(* IEC 61131-3 sources: plcassist-cli/packages/volt-lsp-iec/test-corpus/pro2193/Device/Plc Logic/Application/99 Library/Function Blocks/Modules, 9 files *)

(* ---- LockFB.fb ---- *)
// Use the TEST_AND_SET operator to ensure exclusive access.
{attribute 'no_explicit_call' := 'No need to call this FB. Only the methods are used'}
{attribute 'monitoring_display' := 'currentLockHolder'}
FUNCTION_BLOCK LockFB
VAR
	dwSynch							: DWORD;		// Lock object
	currentLockHolder				: STRING(80);	// Name of the module that is currently locking this FB
	currentLockHolderIsWithoutLock	: BOOL;
END_VAR
VAR_OUTPUT
	callCounter						: UDINT;
END_VAR

END_FUNCTION_BLOCK

// Force releasing the lock
METHOD ForceRelease
Release(currentLockHolder);
END_METHOD

// Release the lock by the current lock holder
METHOD Release : BOOL
VAR_INPUT
	locker		: STRING(80);		// The module that is releasing the lock
END_VAR
IF locker <> currentLockHolder THEN
	RETURN;
END_IF

IF locker <> '' OR dwSynch <> 0 THEN
	LogPlc.Debug(CONCAT5('Lock released by: ', locker, ', lock duration: ', TO_STRING(callCounter), ' PLC cycles'));
END_IF

dwSynch							:= 0;		// The DWORD must be reset to release the lock
currentLockHolder				:= '';		// Clear name of locker
currentLockHolderIsWithoutLock	:= FALSE;
callCounter						:= 0;

Release							:= TRUE;
END_METHOD

// Request a lock. Returns false if the lock is already taken by someone else.
METHOD Request : BOOL
VAR_INPUT
	locker		: STRING(80);		// The module that is requesting the lock
END_VAR
IF currentLockHolder = locker THEN		// Check if already locked by locker
	Request := TRUE;					// Locking succeeded
ELSIF TEST_AND_SET(dwSynch) = 0 THEN	// Write the 1 and read the old value at the same time; Result of 0 means no other task is currently locking this FB
	currentLockHolder := locker;		// Save name of locker
	LogPlc.Debug(CONCAT('Lock granted to: ', locker));
	Request := TRUE;					// Locking succeeded
ELSIF currentLockHolderIsWithoutLock THEN
	currentLockHolder := locker;		// Save name of locker
	LogPlc.Debug(CONCAT('Lock stolen by: ', locker));
	Request := TRUE;					// Locking succeeded
ELSE
	Request := FALSE;					// Locking failed. Allready locked by someone else.
END_IF

IF Request THEN
	callCounter := callCounter + 1;
END_IF
END_METHOD

// Request a lock without actually locking. Use if a command should be overruled by a second command.
{attribute 'obsolete' := 'Do not use! Method makes no sense. See below for discussion'}
METHOD RequestWithoutLock : BOOL
VAR_INPUT
	locker		: STRING(80);		// The module that is requesting the lock
END_VAR

// locking without actually locking makes no sense to me!
// Just NOT lock a command if you don't need a lock.
// If we really need it we could add optional bool parameter to Request method: WeakLock or something
// Stefan 3-7-25
IF currentLockHolder = locker THEN		// Check if already locked by locker
	RequestWithoutLock := TRUE;			// Locking succeeded
ELSIF TEST_AND_SET(dwSynch) = 0 THEN	// Write the 1 and read the old value at the same time; Result of 0 means no other task is currently locking this FB
	currentLockHolder := locker;		// Save name of locker
	LogPlc.Debug(CONCAT('Lock granted to: ', locker));
	currentLockHolderIsWithoutLock := TRUE;
	RequestWithoutLock := TRUE;			// Locking succeeded
ELSIF currentLockHolderIsWithoutLock THEN
	currentLockHolder := locker;		// Save name of locker
	LogPlc.Debug(CONCAT('Lock stolen by: ', locker));
	RequestWithoutLock := TRUE;			// Locking succeeded
ELSE
	RequestWithoutLock := FALSE;		// Locking failed. Allready locked by someone else.
END_IF

IF RequestWithoutLock THEN
	callCounter := callCounter + 1;
END_IF
END_METHOD

// Return true the first cycle that the lock is granted.
PROPERTY PUBLIC FirstCall : BOOL

// No monitoring attribute because property is only high for 1 cycle.
GET
VAR
END_VAR
FirstCall := callCounter = 1;
END_GET
END_PROPERTY

// Return true when a lock is active
{attribute 'monitoring':='call'}
PROPERTY PUBLIC IsLocked : BOOL
GET
VAR
END_VAR
IsLocked := currentLockHolder <> '';
END_GET
END_PROPERTY

(* ---- ModuleBaseHardwareFB.fb ---- *)
// Modules that react to EStop and Stop events from the machine
{attribute 'symbol' := 'none'}
FUNCTION_BLOCK PUBLIC ABSTRACT ModuleBaseHardwareFB
EXTENDS ModuleRegisterableFB
IMPLEMENTS IModuleBase, IModuleWithCommandLock
VAR
	CommandLock					: LockFB;		// Internal lock. Lock hardware unit when a command is active
	ProcessCommandLock			: LockFB;		// External lock from the process. So a process can claim a hardware unit for itself
END_VAR

SUPER^();

Alarms();	// Handle custom alarms that are not defined in the FB's called in Cyclic()

END_FUNCTION_BLOCK

METHOD PROTECTED Alarms
END_METHOD

// Command to reset the module (Statemachine to zero state) in case of E-Stop
METHOD PUBLIC EStop : BOOL	// Returns true when drives are in standstill

(* Command to reset the module (Statemachine to zero state) in case of E-Stop

Add code here to handle emergency stops. For example:

// Reset the state of the unit.
State := MyUnit_State.None;

// Stop the servo drive
Drive.Stop(TRUE);

// Reset all cylinders and outputs
SomeCylinder.Reset();
SomeOtherOutput.Reset();

// Reset all vacuums with a helper function
VacuumResetAll(Vacuum);

// Does this module have a servo drive? Then you can return true when the drive has braked to standstill
EStop := Drive.Standstill OR NOT Drive.AxisEnabled;
// Else, just return true.
EStop := TRUE;

 *)
CommandLock.ForceRelease();
ProcessCommandLock.ForceRelease();

EStop := TRUE;
END_METHOD

// Force releasing the lock
METHOD LockForceRelease
ProcessCommandLock.ForceRelease();
END_METHOD

// Release the lock by the current lock holder
METHOD PUBLIC LockRelease : BOOL
VAR_INPUT
	locker		: STRING(80);		// The module that is releasing the lock
END_VAR
LockRelease		:= ProcessCommandLock.Release(locker);
END_METHOD

// Request a lock. Returns false if the lock is already taken by someone else.
METHOD PUBLIC LockRequest : BOOL
VAR_INPUT
	locker		: STRING(80);		// The module that is requesting the lock
END_VAR
LockRequest		:= ProcessCommandLock.Request(locker);
END_METHOD

// Command to stop a module (Statemachine to zero state)
METHOD PUBLIC Stop : BOOL	// Returns true when drives are in standstill
CommandLock.ForceRelease();
ProcessCommandLock.ForceRelease();

Stop := TRUE;
END_METHOD

(* ---- ModuleManagerFB.fb ---- *)
// Function block to register all modules in the program. So its no longer needed to manually fill an array in the SER program.
{attribute 'no_explicit_call' := 'Do not call this FB. This is just a place to store data about regestered modules.'}
{attribute 'no_assign'}
FUNCTION_BLOCK FINAL ModuleManagerFB
IMPLEMENTS IModuleManager
VAR_OUTPUT
	baseModules				: ARRAY[1..GVL_Constants.MaxNumberOfModules] OF IModuleBase;
	baseModulesCount		: UINT;

	startableModules		: ARRAY[1..GVL_Constants.MaxNumberOfStartableModules] OF IModuleStartable;
	startableModulesCount	: UINT;

	resettableModules		: ARRAY[1..GVL_Constants.MaxNumberOfResettableModules] OF IModuleResettable;
	resettableModulesCount	: UINT;

	servoDrives				: ARRAY[1..GVL_Constants.MaxNumberOfServoDrives] OF IServoDrive;
	servoDrivesCount		: UINT;

	gates					: ARRAY[1..GVL_Constants.MaxNumberOfGates] OF ISafetyGate;
	gatesCount				: UINT;

END_VAR
VAR
	{attribute 'hide'}	_name					: STRING(12);									// Name of module manager
	{attribute 'hide'}	_moduleHandler			: L_IMHP.L_IMHP_ModuleHandler :=				// Lenze module handler
						(
							Layer				:= L_IMHP_Layer.Process_Control,
							CompType			:= L_IMHP_ComponentType.GeneralMachineModule
						);
END_VAR

END_FUNCTION_BLOCK

//FB_Init is always available implicitly and it is used primarily for initialization.
//The return value is not evaluated. For a specific influence, you can also declare the
//methods explicitly and provide additional code there with the standard initialization
//code. You can evaluate the return value.
METHOD FB_Init: BOOL
VAR_INPUT
	bInitRetains	: BOOL;							// TRUE: the retain variables are initialized (reset warm / reset cold)
	bInCopyCode		: BOOL;							// TRUE: the instance will be copied to the copy code afterward (online change)

	name			: STRING(12);					// Give name of module manager (For example SER or BFU)
END_VAR
THIS^._name						:= name;
THIS^._moduleHandler.CompName	:= name;
END_METHOD

METHOD PRIVATE LogMessage
VAR_INPUT
	moduleName		: STRING(12);
	selUnRegister	: BOOL;
	index			: UINT;
	module			: IAbleToRegister;
END_VAR
LogPlc.Debug(
	CONCAT9(
		Name,
		': ',
		moduleName,
		' module ',
		TO_STRING(index),
		SEL(selUnRegister, ' registered: ', ' unregistered: '),
		module.InstanceName,
		SEL(module.MemoryAddress = '', ', Address: ', ''),
		module.MemoryAddress
	)
);
END_METHOD

// Registers a module
METHOD Register : BOOL
VAR_INPUT
	thingToRegister	: IAbleToRegister;
END_VAR
VAR
	baseModule		: IModuleBase;
	startableModule	: IModuleStartable;
	resettableModule: IModuleResettable;
	servoDrive		: IServoDrive;
	gate			: ISafetyGate;

	thingMatchedAnyInterface : BOOL;
END_VAR
IF thingToRegister = 0 THEN
	LogPlc.Fatal('Null reference exception! Interface does not exist.');
	RETURN;
END_IF

IF __QUERYINTERFACE(thingToRegister, baseModule) THEN
	IF baseModulesCount = GVL_Constants.MaxNumberOfModules THEN
		LogPlc.Fatal(CONCAT('Register Full! Module NOT registered: ', thingToRegister.InstanceName));
	ELSE
		thingMatchedAnyInterface				:= TRUE;
		Increment.AnyInt(baseModulesCount);
		baseModules[baseModulesCount]			:= baseModule;
		LogMessage('Base', FALSE, baseModulesCount, thingToRegister);
	END_IF
END_IF

IF __QUERYINTERFACE(thingToRegister, startableModule) THEN
	IF startableModulesCount = GVL_Constants.MaxNumberOfStartableModules THEN
		LogPlc.Fatal(CONCAT('Startable Register Full! Module NOT registered: ', thingToRegister.InstanceName));
	ELSE
		thingMatchedAnyInterface				:= TRUE;
		Increment.AnyInt(startableModulesCount);
		startableModules[startableModulesCount]	:= startableModule;
		LogMessage('Startable', FALSE, startableModulesCount, thingToRegister);
	END_IF
END_IF

IF __QUERYINTERFACE(thingToRegister, resettableModule) THEN
	IF resettableModulesCount = GVL_Constants.MaxNumberOfResettableModules THEN
		LogPlc.Fatal(CONCAT('Resettable Register Full! Module NOT registered: ', thingToRegister.InstanceName));
	ELSE
		thingMatchedAnyInterface				:= TRUE;
		Increment.AnyInt(resettableModulesCount);
		resettableModules[resettableModulesCount] := resettableModule;
		LogMessage('Resettable', FALSE, resettableModulesCount, thingToRegister);
	END_IF
END_IF

IF __QUERYINTERFACE(thingToRegister, servoDrive) THEN
	IF servoDrivesCount = GVL_Constants.MaxNumberOfServoDrives THEN
		LogPlc.Fatal(CONCAT('Servodrive Register Full! Module NOT registered: ', thingToRegister.InstanceName));
	ELSE
		thingMatchedAnyInterface				:= TRUE;
		Increment.AnyInt(servoDrivesCount);
		servoDrives[servoDrivesCount]			:= servoDrive;
		LogMessage('Servo', FALSE, servoDrivesCount, thingToRegister);
	END_IF
END_IF

IF __QUERYINTERFACE(thingToRegister, gate) THEN
	IF gatesCount = GVL_Constants.MaxNumberOfGates THEN
		LogPlc.Fatal(CONCAT('Gate Register Full! Module NOT registered: ', thingToRegister.InstanceName));
	ELSE
		thingMatchedAnyInterface				:= TRUE;
		Increment.AnyInt(gatesCount);
		gates[gatesCount]						:= gate;
		LogMessage('Gate', FALSE, gatesCount, thingToRegister);
	END_IF
END_IF

IF NOT thingMatchedAnyInterface THEN
	LogPlc.Fatal(Concat('Unable to register module: ', thingToRegister.InstanceName));	// Please add a handler for this kind of interface
END_IF

Register := TRUE;
END_METHOD

// Unregisters a module
METHOD Unregister : BOOL
VAR_INPUT
	thingToRegister	: IAbleToRegister;
END_VAR
VAR
	i				: UINT;
	moduleIndex		: UINT;
	baseModule		: IModuleBase;
	startableModule	: IModuleStartable;
	resettableModule: IModuleResettable;
	servoDrive		: IServoDrive;
	gate			: ISafetyGate;
	thingMatchedAnyInterface : BOOL;
END_VAR
IF thingToRegister = 0 THEN
	LogPlc.Fatal('Null reference exception! Interface does not exist.');
	RETURN;
END_IF

// Check if the current interface is of type: module
IF __QUERYINTERFACE(thingToRegister, baseModule) THEN
	FOR i := 1 TO GVL_Constants.MaxNumberOfModules DO
		IF baseModule = baseModules[i] THEN		// Find the module in the register
			moduleIndex := i;				// Store location where it was found
			baseModules[i] := 0;			// Clear the reference
			baseModulesCount := baseModulesCount - 1;	// Decrease count
			LogMessage('Base', TRUE, moduleIndex, thingToRegister);
			EXIT;
		END_IF
	END_FOR
	// Move all references in the register one place up, so there are no gaps in the array.
	IF moduleIndex > 0 AND moduleIndex < GVL_Constants.MaxNumberOfModules THEN
		FOR i := moduleIndex TO GVL_Constants.MaxNumberOfModules - 1 DO
			baseModules[i] := baseModules[i + 1];
			IF baseModules[i + 1] = 0 THEN
				EXIT;
			END_IF
		END_FOR
	END_IF
	thingMatchedAnyInterface := TRUE;
	moduleIndex := 0;
END_IF

IF __QUERYINTERFACE(thingToRegister, startableModule) THEN
	FOR i := 1 TO GVL_Constants.MaxNumberOfStartableModules DO
		IF startableModule = startableModules[i] THEN
			moduleIndex := i;
			startableModules[i] := 0;
			startableModulesCount := startableModulesCount - 1;
			LogMessage('Startable', TRUE, moduleIndex, thingToRegister);
			EXIT;
		END_IF
	END_FOR
	IF moduleIndex > 0 AND moduleIndex < GVL_Constants.MaxNumberOfStartableModules THEN
		FOR i := moduleIndex TO GVL_Constants.MaxNumberOfStartableModules - 1 DO
			startableModules[i] := startableModules[i + 1];
			IF startableModules[i + 1] = 0 THEN
				EXIT;
			END_IF
		END_FOR
	END_IF
	thingMatchedAnyInterface := TRUE;
	moduleIndex := 0;
END_IF

IF __QUERYINTERFACE(thingToRegister, resettableModule) THEN
	FOR i := 1 TO GVL_Constants.MaxNumberOfResettableModules DO
		IF resettableModule = resettableModules[i] THEN
			moduleIndex := i;
			resettableModules[i] := 0;
			resettableModulesCount := resettableModulesCount - 1;
			LogMessage('Resettable', TRUE, moduleIndex, thingToRegister);
			EXIT;
		END_IF
	END_FOR
	IF moduleIndex > 0 AND moduleIndex < GVL_Constants.MaxNumberOfResettableModules THEN
		FOR i := moduleIndex TO GVL_Constants.MaxNumberOfResettableModules - 1 DO
			resettableModules[i] := resettableModules[i + 1];
			IF resettableModules[i + 1] = 0 THEN
				EXIT;
			END_IF
		END_FOR
	END_IF
	thingMatchedAnyInterface := TRUE;
	moduleIndex := 0;
END_IF

IF __QUERYINTERFACE(thingToRegister, servoDrive) THEN
	FOR i := 1 TO GVL_Constants.MaxNumberOfServoDrives DO
		IF servoDrive = servoDrives[i] THEN
			moduleIndex := i;
			servoDrives[i] := 0;
			servoDrivesCount := servoDrivesCount - 1;
			LogMessage('Servo', TRUE, moduleIndex, thingToRegister);
			EXIT;
		END_IF
	END_FOR
	IF moduleIndex > 0 AND moduleIndex < GVL_Constants.MaxNumberOfServoDrives THEN
		FOR i := moduleIndex TO GVL_Constants.MaxNumberOfServoDrives - 1 DO
			servoDrives[i] := servoDrives[i + 1];
			IF servoDrives[i + 1] = 0 THEN
				EXIT;
			END_IF
		END_FOR
	END_IF
	thingMatchedAnyInterface := TRUE;
	moduleIndex := 0;
END_IF

IF __QUERYINTERFACE(thingToRegister, gate) THEN
	FOR i := 1 TO GVL_Constants.MaxNumberOfGates DO
		IF gate = gates[i] THEN
			moduleIndex := i;
			gates[i] := 0;
			gatesCount := gatesCount - 1;
			LogMessage('Gate', TRUE, moduleIndex, thingToRegister);
			EXIT;
		END_IF
	END_FOR
	IF moduleIndex > 0 AND moduleIndex < GVL_Constants.MaxNumberOfGates THEN
		FOR i := moduleIndex TO GVL_Constants.MaxNumberOfGates - 1 DO
			gates[i] := gates[i + 1];
			IF gates[i + 1] = 0 THEN
				EXIT;
			END_IF
		END_FOR
	END_IF
	thingMatchedAnyInterface := TRUE;
	moduleIndex := 0;
END_IF

IF NOT thingMatchedAnyInterface THEN
	LogPlc.Fatal(Concat('Unable to unregister module: ', thingToRegister.InstanceName));	// Please add a handler for this kind of interface
END_IF

Unregister := TRUE;
END_METHOD

PROPERTY PUBLIC ModuleHandler : L_IMHP.L_IMHP_IModuleHandler
GET
VAR
END_VAR
ModuleHandler	:= _moduleHandler;
END_GET
END_PROPERTY

PROPERTY PUBLIC Name : STRING(12)
GET
VAR
END_VAR
Name	:= _name;

// This does not work because CompName has no Getter. Maybe change in the future when Lenze changes library
// Name	:= _moduleHandler.CompName;
END_GET
END_PROPERTY

(* ---- ModuleRegisterableFB.fb ---- *)
// Module registers itself with central module manager. Also implements Lenze module manager
{attribute 'reflection'}
{attribute 'monitoring_display' := '_instanceName'}
{attribute 'symbol' := 'none'}
FUNCTION_BLOCK PUBLIC ABSTRACT ModuleRegisterableFB
IMPLEMENTS IAbleToRegister
VAR
	ModuleManager				: IModuleManager;				// Location of module manager where this module is stored
	ModuleHandler				: L_IMHP.L_IMHP_ModuleHandler;	// Lenze module handler (No need to call this FB)

	{attribute 'hide'}
	{attribute 'no_copy'}
	_instanceNo					: UINT;				// Private backing field for instance number (start from 1)
	{attribute 'instance-path'}
	{attribute 'noinit'}
	{attribute 'hide'}
	_instanceName				: STRING(80);		// Private backing field for instance name (automatically generated by compiler)

	{attribute 'no_copy'}
	ModuleParent				: L_IMHP.L_IMHP_IModuleHandler;

	{attribute 'hide'}
	{attribute 'init_on_onlchange'}
	_initialized				: BOOL	:= FALSE;	// Is high when init is done
END_VAR
VAR_STAT
	moduleCurrentlyExecuting	: STRING(80);		// For debugging: In case of exception check this string to see what module is currently executing
END_VAR

IF NOT _initialized THEN
	_initialized := TRUE;
	Initialize();
END_IF

stu.StrCpyA(
	pBuffer		:= ADR(moduleCurrentlyExecuting),
	iBufferSize	:= SIZEOF(moduleCurrentlyExecuting),
	pStr		:= ADR(_instanceName)
	);

Cyclic();	// Do stuff every PLC cycle (like instantiate all fbs needed in the module).

END_FUNCTION_BLOCK

METHOD PROTECTED Cyclic
END_METHOD

//FB_Exit must be implemented explicitly. If there is an implementation, then the
//method is called before the controller removes the code of the function block instance
//(implicit call). The return value is not evaluated.
METHOD FB_Exit: BOOL
VAR_INPUT
	bInCopyCode: BOOL;  // TRUE: the exit method is called in order to leave the instance which will be copied afterwards (online change).
END_VAR
IF THIS^.ModuleManager <> 0 THEN
	THIS^.ModuleManager.Unregister(THIS^);
END_IF

THIS^.ModuleParent	:= 0;
END_METHOD

//FB_Init is always available implicitly and it is used primarily for initialization.
//The return value is not evaluated. For a specific influence, you can also declare the
//methods explicitly and provide additional code there with the standard initialization
//code. You can evaluate the return value.
METHOD FB_Init: BOOL
VAR_INPUT
	bInitRetains	: BOOL;							// TRUE: the retain variables are initialized (reset warm / reset cold)
	bInCopyCode		: BOOL;							// TRUE: the instance will be copied to the copy code afterward (online change)

	instanceNo		: UINT;
	moduleManager	: IModuleManager;				// Give location of module manager (can be different for SER or BFU)
	moduleParent	: L_IMHP.L_IMHP_IModuleHandler;	// (Optional) Give parent of this module. Use zero to use SER or BFU as parent.
END_VAR
THIS^.ModuleManager		:= moduleManager;

IF moduleManager = 0 THEN
	LogPlc.Info(CONCAT(_instanceName, ' has no module manager to register to. Is this intended?'));
ELSE
	moduleManager.Register(THIS^);		// Register this module with the central module manager.
END_IF

IF moduleParent <> 0 THEN
	THIS^.ModuleParent	:= moduleParent;
ELSIF moduleManager <> 0 THEN
	THIS^.ModuleParent	:= moduleManager.ModuleHandler;
END_IF

// Set instance number
IF instanceNo = 0 THEN
	LogPlc.Fatal(CONCAT(_instanceName, ' has instanceNo 0. Use instanceNo > 0.'));
END_IF

_instanceNo				:= instanceNo;

ParseInstanceName(ADR(_instanceName));

ModuleHandler.CompName	:= InstanceName;
ModuleHandler.Layer		:= L_IMHP_Layer.Tech_Application;
ModuleHandler.CompType	:= L_IMHP_ComponentType.GeneralMachineModule;

// Warning: Only when module is of CompType = MachineModule or GeneralMachineModule, are active alarms kicked up to the parent module!
END_METHOD

METHOD PROTECTED Initialize
ModuleHandler.SetParent(
					ModuleHandlerParent	:= ModuleParent,
					RelationShip		:= L_IMHP.L_IMHP_RelationshipID.ApplicationView);
END_METHOD

// Automatically generated name of the instance
{attribute 'monitoring':='call'}
PROPERTY PUBLIC InstanceName : STRING(80)
GET
VAR
END_VAR
InstanceName := _instanceName;
END_GET
END_PROPERTY

// Instance number, the number of the module or unit (start from 1)
{attribute 'monitoring':='call'}
PROPERTY PUBLIC InstanceNo : UINT

// Note: this number does not have to be unique for each module...
GET
VAR
END_VAR
InstanceNo := _instanceNo;
END_GET
END_PROPERTY

// Location of the FB in memory (for debugging)
{attribute 'monitoring':='call'}
PROPERTY PUBLIC MemoryAddress : STRING(8)
GET
VAR
END_VAR
{IF defined (IsSimulationMode)}
	MemoryAddress := DWORD_TO_HEXSTRING(TO_DWORD(ADR(THIS^)));
{ELSE}
	MemoryAddress := '';
{END_IF}
END_GET
END_PROPERTY

(* ---- ModuleResettableFB.fb ---- *)
// Generic variables that all modules use
{attribute 'symbol' := 'none'}
FUNCTION_BLOCK PUBLIC ABSTRACT ModuleResettableFB
EXTENDS ModuleBaseHardwareFB
IMPLEMENTS IModuleResettable
VAR
	{attribute 'hide'}
	{attribute 'no_copy'}
	_resetConditions			: ARRAY[1..2] OF IModuleResettable;
END_VAR

SUPER^();

END_FUNCTION_BLOCK

//FB_Init is always available implicitly and it is used primarily for initialization.
//The return value is not evaluated. For a specific influence, you can also declare the
//methods explicitly and provide additional code there with the standard initialization
//code. You can evaluate the return value.
{attribute 'analysis' := '-33'}
METHOD FB_Init: BOOL
VAR_INPUT
	bInitRetains	: BOOL;							// TRUE: the retain variables are initialized (reset warm / reset cold)
	bInCopyCode		: BOOL;							// TRUE: the instance will be copied to the copy code afterward (online change)

	instanceNo		: UINT;							// Handled in ModuleRegisterableFB.FB_Init method
	moduleManager	: IModuleManager;				// Handled in ModuleRegisterableFB.FB_Init method
	moduleParent	: L_IMHP.L_IMHP_IModuleHandler;	// Handled in ModuleRegisterableFB.FB_Init method

	resetCondition1	: IModuleResettable;
	resetCondition2	: IModuleResettable;
END_VAR
_resetConditions[1]	:= resetCondition1;
_resetConditions[2]	:= resetCondition2;
END_METHOD

// Command to reset the module. Servodrives are homed.
METHOD PUBLIC ABSTRACT Reset : BOOL	// Returns true when homing done
END_METHOD

// The order in which the modules are homed.
{attribute 'monitoring':='call'}
PROPERTY PUBLIC ResetCondition1 : IModuleResettable
GET
VAR
END_VAR
ResetCondition1	:= _resetConditions[1];
END_GET
END_PROPERTY

// The order in which the modules are homed.
{attribute 'monitoring':='call'}
PROPERTY PUBLIC ResetCondition2 : IModuleResettable
GET
VAR
END_VAR
ResetCondition2	:= _resetConditions[2];
END_GET
END_PROPERTY

(* ---- ModuleWithBrakedServoBaseFB.fb ---- *)
// Extra variables for modules that have a servo drive
{attribute 'symbol' := 'none'}
FUNCTION_BLOCK PUBLIC ABSTRACT ModuleWithBrakedServoBaseFB
EXTENDS ModuleWithServoBaseFB
VAR_INPUT
	ButtonReleaseBrake			: PushButtonLedFB;
END_VAR
VAR
	{attribute 'symbol' := 'read'}	DriveBrakeLogic				: ServoDriveBrakeLogicFB;
END_VAR

SUPER^(
	AxisRef				:= AxisRef,
	DataBrink			:= DataBrink,
	coveredDistance		:= coveredDistance,
);

ButtonReleaseBrake();

DriveBrakeLogic(
	AxisRef				:= AxisRef,
	xBrakeReleaseIn		:= ButtonReleaseBrake.buttonInput);

END_FUNCTION_BLOCK

(* ---- ModuleWithServoBaseFB.fb ---- *)
// Extra variables for modules that have a servo drive
{attribute 'symbol' := 'none'}
FUNCTION_BLOCK PUBLIC ABSTRACT ModuleWithServoBaseFB
EXTENDS ModuleResettableFB
IMPLEMENTS IModuleManualControlEnabled
VAR_INPUT
	xEnableServoDrive			: BOOL;
	xQuickStop					: BOOL;
END_VAR
VAR_IN_OUT
	AxisRef						: L_MC1P.AXIS_REF;
	DataBrink					: DataBrinkType;
	coveredDistance				: UDINT;
END_VAR
VAR
	{attribute 'symbol' := 'read'}	Drive						: ServoDriveFB
	(
		instanceNo		:= 1,
		moduleManager	:= ModuleManager,
		moduleParent	:= ModuleHandler,
	);

	// Forward alarms of children (ServoDriveFB) to parent
	ForwardSeverity				: L_IE1P.L_IE1P_ForwardSeverity;

	// Manual control of servo drive is enabled from outside this module
	externalManualServoControlEnabled		: BOOL;
	// Manual control of servo drive is enabled from inside the module
	internalManualServoControlEnabled		: BOOL := TRUE;

	ManualControlIsBlockedWarning			: ARRAY[1..6] OF SetErrorFB;

END_VAR

SUPER^();

Drive(
	globalSpeedOverride			:= PersistentVars.usiGlobalSERSpeed,
	globalSpeedOverrideEnable	:= ,
	rSetManualSpeed				:= 5,
	xGlobalReset				:= GlobalVars.Reset,
	xEnableDrive				:= xEnableServoDrive,
	xQuickStop					:= xQuickStop,
	manualControlEnabled		:= SER.ManualControlEnabled
								AND Drive.AxisEnabled
								AND externalManualServoControlEnabled
								AND internalManualServoControlEnabled
								AND PNOZMulti2.xHoldToRunButton,
	servoJogMode				:= HMI.servoJogMode,
	AxisRef						:= AxisRef,
	DataBrink					:= DataBrink,
	coveredDistance				:= coveredDistance);

ForwardSeverity(
	xEnable						:= TRUE,
	ModuleHandler				:= ModuleHandler,
	xForwardFromChildModules	:= TRUE,
	xDisableForwardToParent		:= ,
	xBusy						=> ,
	xError						=> ,
	eErrorID					=> );

ManualControlIsBlockedWarning[1](
	moduleHandler	:= ModuleHandler,
	textRefId		:= General_Unit_Errors,
	errorId			:= 6,
	alarmCondition	:= Drive.manualControlIsBlocked AND NOT SER.ManualControlEnabled,
	alarmDelay		:= 0.0,
	severity		:= enumErrorSeverity.Warning_Lock,
	reaction		:= enumErrorReaction.No_reaction);

ManualControlIsBlockedWarning[2](
	moduleHandler	:= ModuleHandler,
	textRefId		:= General_Unit_Errors,
	errorId			:= 7,
	alarmCondition	:= Drive.manualControlIsBlocked AND NOT Drive.AxisEnabled,
	alarmDelay		:= 0.0,
	severity		:= enumErrorSeverity.Warning_Lock,
	reaction		:= enumErrorReaction.No_reaction);

ManualControlIsBlockedWarning[3](
	moduleHandler	:= ModuleHandler,
	textRefId		:= General_Unit_Errors,
	errorId			:= 8,
	alarmCondition	:= Drive.manualControlIsBlocked AND NOT externalManualServoControlEnabled,
	alarmDelay		:= 0.0,
	severity		:= enumErrorSeverity.Warning_Lock,
	reaction		:= enumErrorReaction.No_reaction);

ManualControlIsBlockedWarning[4](
	moduleHandler	:= ModuleHandler,
	textRefId		:= General_Unit_Errors,
	errorId			:= 9,
	alarmCondition	:= Drive.manualControlIsBlocked AND NOT internalManualServoControlEnabled,
	alarmDelay		:= 0.0,
	severity		:= enumErrorSeverity.Warning_Lock,
	reaction		:= enumErrorReaction.No_reaction);

ManualControlIsBlockedWarning[5](
	moduleHandler	:= ModuleHandler,
	textRefId		:= General_Unit_Errors,
	errorId			:= 10,
	alarmCondition	:= Drive.manualControlIsBlocked AND NOT PNOZMulti2.xHoldToRunButton,
	alarmDelay		:= 0.0,
	severity		:= enumErrorSeverity.Warning_Lock,
	reaction		:= enumErrorReaction.No_reaction);

ManualControlIsBlockedWarning[6](
	moduleHandler	:= ModuleHandler,
	textRefId		:= General_Unit_Errors,
	errorId			:= 11,
	alarmCondition	:= Drive.manualControlIsBlocked AND Drive.AxisBasicControl.xInternalControlActive,
	alarmDelay		:= 0.0,
	severity		:= enumErrorSeverity.Warning_Lock,
	reaction		:= enumErrorReaction.No_reaction);

END_FUNCTION_BLOCK

METHOD PROTECTED Initialize
SUPER^.Initialize();

Drive.config.axisBlockedAlarmMaxTorque	:= 0.5;
END_METHOD

// Manual control of hardware is enabled from external context
{attribute 'monitoring':='call'}
PROPERTY ExternalManualControlEnabled : BOOL
SET
VAR
END_VAR
externalManualServoControlEnabled := ExternalManualControlEnabled;
END_SET
END_PROPERTY

(* ---- ModuleWithStateFB.fb ---- *)
// Modules that have a state (Processes). Keep a history with StateMachineHistoryFB
{attribute 'symbol' := 'none'}
FUNCTION_BLOCK PUBLIC ABSTRACT ModuleWithStateFB
EXTENDS ModuleRegisterableFB
IMPLEMENTS IModuleBase
VAR
	CommandLock					: LockFB;		// Internal lock. Lock hardware unit when a command is active (check if we can remove this!! Processes do not need locks ?? SR)

	{attribute 'symbol' := 'read'}	State	: StateMachineHistoryFB(instanceName:= InstanceName);		// Call this FB in Cyclic() in your Process module!

	{attribute 'hide'}	noProgramWarningBusy		: BIT;
	{attribute 'hide'}	noProgramWarningDone		: BIT;
END_VAR

SUPER^();

noProgramWarningDone R= NOT noProgramWarningBusy;
noProgramWarningBusy := FALSE;

// Execute state machine of module
Execute();

END_FUNCTION_BLOCK

METHOD PROTECTED ABSTRACT Cyclic

// Modules with a State must have a Cyclic method: to call State FB
END_METHOD

// Command to reset the module (Statemachine to zero state) in case of E-Stop
METHOD PUBLIC ABSTRACT EStop : BOOL	// Returns true when drives are in standstill

(* Command to reset the module (Statemachine to zero state) in case of E-Stop

Add code here to handle emergency stops. For example:

// Reset the state of the unit.
State := MyUnit_State.None;

// Stop the servo drive
Drive.Stop(TRUE);

// Reset all cylinders and outputs
SomeCylinder.Reset();
SomeOtherOutput.Reset();

// Reset all vacuums with a helper function
VacuumResetAll(Vacuum);

// Does this module have a servo drive? Then you can return true when the drive has braked to standstill
EStop := Drive.Standstill OR NOT Drive.AxisEnabled;
// Else, just return true.
EStop := TRUE;

 *)
END_METHOD

// After a state change, this method is called to execute the current state
METHOD PROTECTED ABSTRACT Execute
END_METHOD

// Here is the State Machine for the default exchangeset
METHOD PROTECTED ABSTRACT Execute_Sequence1
END_METHOD

// Logs a warning in the PLC log when there is a module that has not defined a program for an exchange set.
METHOD PROTECTED ShowNoProgramWarning
// Only write the log message once, the first time the method is executed.
IF NOT noProgramWarningDone THEN
	LogPlc.Warn(CONCAT3(InstanceName, ': No program for: ', TO_STRING(PersistentVars.RecipeVars.ActiveExchangeSet)));
END_IF

noProgramWarningBusy := TRUE;
noProgramWarningDone := TRUE;
END_METHOD

// Command to stop a module (Statemachine to zero state)
METHOD PUBLIC ABSTRACT Stop : BOOL	// Returns true when drives are in standstill
END_METHOD

(* ---- StateMachineHistoryFB.fb ---- *)
{attribute 'symbol' := 'none'}
FUNCTION_BLOCK INTERNAL FINAL StateMachineHistoryFB
EXTENDS MonitoringAddLogBase
VAR_INPUT
	{attribute 'symbol' := 'read'}	actState			: DINT;
END_VAR
VAR_OUTPUT
	StateHistory				: ARRAY[0..HistorySize] OF StateHistoryItemType;	// StateHistory[0] holds previous state
END_VAR
VAR//VISU
	{attribute 'symbol' := 'read'}	timeActive			: REAL;
	{attribute 'symbol' := 'read'}	timeIdle			: REAL;
	{attribute 'symbol' := 'read'}	durationInState		: REAL;						// Duration how long the current state is active.
	{attribute 'symbol' := 'read'}	actStateColor		: enumColorList;			// Color of active tile in HMI
END_VAR
VAR
	{attribute 'hide'}		i							: INT;
	{attribute 'hide'}		prevState					: DINT			:= GVL_Constants.DintSmallest;
	{attribute 'hide'}		timeLastStateTransition		: TIME_OF_DAY	:= TimeSettings.todNow;
	{attribute 'hide'}		instanceName				: STRING(80);
	{attribute 'hide'}		_stateChanged				: BOOL;

	{attribute 'hide'}		CycleTimeActive				: MeasureTime;				// Measure cycle times of this module
	{attribute 'hide'}		CycleTimeIdle				: MeasureTime;				// Measure cycle times of this module
	{attribute 'hide'}		measureDuration				: MeasureTime;

	timeout1_Warn_Delay			: REAL			:= 5.0;						// Color tile with warning color when state takes this long
	timeout2_Error_Delay		: REAL			:= 10.0;					// Color tile with error color when state takes this long
	timeout3_Fatal_Delay		: REAL			:= 15.0;					// Color tile with fatal color when state takes this long
	timeout1_Warn_Color			: enumColorList	:= enumColorList.Yellow;	// Warning color for tile
	timeout2_Error_Color		: enumColorList	:= enumColorList.Orange;	// Error color for tile
	timeout3_Fatal_Color		: enumColorList	:= enumColorList.Red;		// Fatal color for tile
END_VAR
VAR CONSTANT
	HistorySize					: INT := 19;
END_VAR

// Measure cycle times
timeIdle		:= CycleTimeActive.Measure(	In := actState < 10);
timeActive		:= CycleTimeIdle.Measure(	In := actState >= 10);
durationInState	:= measureDuration.Measure(	In := TRUE);	// Measure the duration how long the current step is active. Give the tile a color when it takes too long.

// Set color for tiles in HMI
IF actState < 10 THEN		// States 0 - 9 are idle states. Machine can stay in these states without timeouts
	actStateColor	:= enumColorList.Lime;
ELSIF durationInState > timeout3_Fatal_Delay THEN
	actStateColor	:= timeout3_Fatal_Color;
ELSIF durationInState > timeout2_Error_Delay THEN
	actStateColor	:= timeout2_Error_Color;
ELSIF durationInState > timeout1_Warn_Delay THEN
	actStateColor	:= timeout1_Warn_Color;
ELSE
	actStateColor	:= enumColorList.Lime;
END_IF

_stateChanged		:= FALSE;

// Check if act state is different than previous state
IF actState = prevState THEN
	RETURN;
END_IF

// Save a history of states
FOR i := HistorySize TO 1 BY -1 DO
	StateHistory[i]	:= StateHistory[i-1];
END_FOR

StateHistory[0].stateNumber			:= prevState;
StateHistory[0].durationInState		:= durationInState;
StateHistory[0].timeEnterState		:= timeLastStateTransition;
StateHistory[0].timeExitState		:= TimeSettings.todNow;

measureDuration.Measure(In := FALSE);
durationInState := 0;

// Save the time of the last state change
timeLastStateTransition	:= TimeSettings.todNow;

IF GlobalVars.EnableLoggingAllStateChanges THEN
	LogPlc.Info(CONCAT5(instanceName, ' changed state: ', TO_STRING(prevState), ' -> ', TO_STRING(actState)));
END_IF

// Output data to monitoring system (optional)
CallAddLogLINT(actState);

// Save previous state
prevState			:= actState;
_stateChanged		:= TRUE;

END_FUNCTION_BLOCK

//FB_Init is always available implicitly and it is used primarily for initialization.
//The return value is not evaluated. For a specific influence, you can also declare the
//methods explicitly and provide additional code there with the standard initialization
//code. You can evaluate the return value.
METHOD FB_Init: BOOL
VAR_INPUT
	bInitRetains: BOOL; // TRUE: the retain variables are initialized (reset warm / reset cold)
	bInCopyCode: BOOL;  // TRUE: the instance will be copied to the copy code afterward (online change)

	instanceName : STRING(80);		// Private backing field for instance name (automatically generated by compiler)
END_VAR
THIS^.instanceName := instanceName;
END_METHOD

// A tile will turn orange after 10 seconds by default. Use this method to change these default values.
METHOD PUBLIC OverrideDefaultErrorTimeout
VAR_INPUT
	delay		: REAL;
	color		: enumColorList;
END_VAR
%FOLDER Override methods
timeout2_Error_Delay		:= delay;
timeout2_Error_Color		:= color;
END_METHOD

// A tile will turn red after 15 seconds by default. Use this method to change these default values.
METHOD PUBLIC OverrideDefaultFatalTimeout
VAR_INPUT
	delay		: REAL;
	color		: enumColorList;
END_VAR
%FOLDER Override methods
timeout3_Fatal_Delay		:= delay;
timeout3_Fatal_Color		:= color;
END_METHOD

// A tile will switch colors after 5 and 10 and 15 seconds. Use this method to change these default values.
METHOD PUBLIC OverrideDefaultTimeouts
VAR_INPUT
	warningDelay	: REAL;
	errorDelay		: REAL;
	fatalDelay		: REAL;
END_VAR
%FOLDER Override methods
timeout1_Warn_Delay			:= warningDelay;
timeout2_Error_Delay		:= errorDelay;
timeout3_Fatal_Delay		:= fatalDelay;
END_METHOD

// A tile will turn yellow after 5 seconds by default. Use this method to change these default values.
METHOD PUBLIC OverrideDefaultWarningTimeout
VAR_INPUT
	delay		: REAL;
	color		: enumColorList;
END_VAR
%FOLDER Override methods
timeout1_Warn_Delay			:= delay;
timeout1_Warn_Color			:= color;
END_METHOD

// Trigger boolean when a state changes
PROPERTY PUBLIC Changed : BOOL
//{attribute 'monitoring':='call'}	No monitoring because property is true for a single plc cycle
GET
VAR
END_VAR
Changed := _stateChanged;
END_GET
END_PROPERTY
